PROGRAM MAIN
VAR

	fbLogHandler : FB_LogHandler;
	
END_VAR


fbLogHandler();

// Run the Diagnostics PRG
//DIAGNOSTICS();

(* FEE devices*)
PRG_FEE();
PRG_Hutch_Gauges();
//PRG_Hutch_Beamline_Valves();
PRG_Roughing_Pumps();

PMPS();

END_PROGRAM

(* stored: Version 1.1.0.1, ProductVersion 3.1.4022.18
   POU MAIN: Id {53e436ba-9af9-4ca4-ad7b-a6b2399fa417}, SpecialFunc None *)
